# EPICS substitutions: db/music_hv_FHF1.substitutions
#
# i.keshelashvili@gsi.de
#
file "db/music_hv.template"
{
     pattern
    {
        FC,  CH
    }

    {
        1, 0
        2, 1
        3, 2
    }
}
